// TIA Portal project "PLC1500与G120调速控制" (V14)

(* hardware
DEVICE "S71500/ET200MP station_1"  S7-1500 station
   slot 0: "导轨_0"  Rack  6ES7 590-1***0-0AA0
   slot 1: "Line1_Station1_PLC"  CPU 1516-3 PN/DP  6ES7 516-3AN01-0AB0  V2.1
      slot 3: "CPU 显示_1"  6ES7591-1BA00-0AA0
   slot 2: "DI 32x24VDC HF_1"  DI 32x24VDC HF  6ES7 521-1BL00-0AB0  V2.1
   slot 3: "DQ 32x24VDC/0.5A HF_1"  DQ 32x24VDC/0.5A HF  6ES7 522-1BL01-0AB0  V1.0
   slot 4: "AI 8xU/I/RTD/TC ST_1"  AI 8xU/I/RTD/TC ST  6ES7 531-7KF00-0AB0  V2.1
   slot 5: "AQ 4xU/I ST_1"  AQ 4xU/I ST  6ES7 532-5HD00-0AB0  V2.1
DEVICE "SINAMICS G_1"  Sinamics.Device
   slot 0: "Line1_Station1_G120"  G120 CU250S-2 PN Vector  6SL3246-0BA22-1FA0  4.7.6
   slot 0: "	_0"  Rail
   slot 3: "PM240-2 IP20"  PM240-2 IP20  6SL3210-1PB13-0ULx  -
*)

// ===== PLC "Line1_Station1_PLC"  CPU 1516-3 PN/DP =====

VAR_GLOBAL   // PLC tag table "默认变量表"
   "状态字" AT %IW256 : Word;   // 变频器反馈的状态
   "速度反馈值" AT %IW258 : Word;   // 变频器当前的速度
   "控制字" AT %QW256 : Word;   // PLC控制变频器内容
   "速度设定值" AT %QW258 : Word;   // PLC控制变频器速度
END_VAR

DATA_BLOCK "通讯控制数据"   // DB1
{ S7_Optimized_Access := 'TRUE' }
VERSION : 0.1
   VAR
      启动 : Bool;   // 用于控制驱动启动
      停止 : Bool;   // 用于控制驱动停止
      反转 : Bool;
      复位 : Bool;
      速度反馈值 : Real;   // 用于存放速度反馈值
      速度设定值 : Real;   // 用于存放速度设定值
      临时变量1 : Real;   // 用于过程数据处理临时存放
      临时变量2 : Real;   // 用于过程数据处理临时存放
      临时变量3 : Real;   // 用于过程数据处理临时存放
      临时变量4 : Real;   // 用于过程数据处理临时存放
   END_VAR
BEGIN
END_DATA_BLOCK

ORGANIZATION_BLOCK "Main"   // OB1, LAD, ProgramCycle
TITLE = "Main Program Sweep (Cycle)"
{ S7_Optimized_Access := 'TRUE' }
VERSION : 0.1
   VAR_INPUT
      Initial_Call : Bool;   // Initial call of this OB
      Remanence : Bool;   // =True, if remanent data are available
   END_VAR
BEGIN

REGION Network 1: 启动程序
   // 启动时,把16#047F写到通讯报文控制字
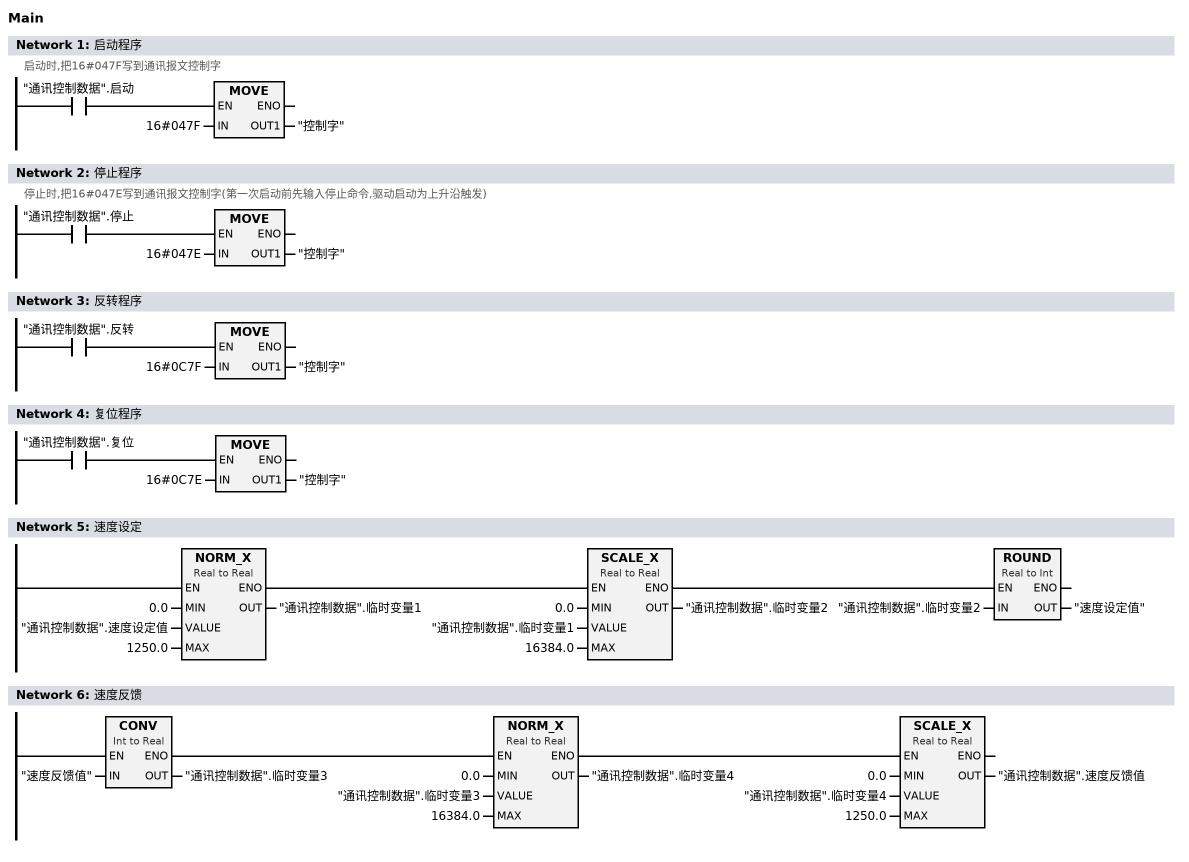
   RUNG wire#powerrail
      Contact( "通讯控制数据".启动 )
      Move(in := 16#047F, out1 => "控制字")
   END_RUNG
   // the same network as SCL:
   IF "通讯控制数据".启动 THEN "控制字" := 16#047F; END_IF;
END_REGION

REGION Network 2: 停止程序
   // 停止时,把16#047E写到通讯报文控制字(第一次启动前先输入停止命令,驱动启动为上升沿触发)
   RUNG wire#powerrail
      Contact( "通讯控制数据".停止 )
      Move(in := 16#047E, out1 => "控制字")
   END_RUNG
   // the same network as SCL:
   IF "通讯控制数据".停止 THEN "控制字" := 16#047E; END_IF;
END_REGION

REGION Network 3: 反转程序
   RUNG wire#powerrail
      Contact( "通讯控制数据".反转 )
      Move(in := 16#0C7F, out1 => "控制字")
   END_RUNG
   // the same network as SCL:
   IF "通讯控制数据".反转 THEN "控制字" := 16#0C7F; END_IF;
END_REGION

REGION Network 4: 复位程序
   RUNG wire#powerrail
      Contact( "通讯控制数据".复位 )
      Move(in := 16#0C7E, out1 => "控制字")
   END_RUNG
   // the same network as SCL:
   IF "通讯控制数据".复位 THEN "控制字" := 16#0C7E; END_IF;
END_REGION

REGION Network 5: 速度设定
   RUNG wire#powerrail
      { S7_Templates := "[SrcType := Real, DestType := Real]" } Normalize(min := 0.0, value := "通讯控制数据".速度设定值, max := 1250.0, out => "通讯控制数据".临时变量1)
      { S7_Templates := "[SrcType := Real, DestType := Real]" } Scale(min := 0.0, value := "通讯控制数据".临时变量1, max := 16384.0, out => "通讯控制数据".临时变量2)
      { S7_Templates := "[SrcType := Real, DestType := Int]" } Round(in := "通讯控制数据".临时变量2, out => "速度设定值")
   END_RUNG
   // the same network as SCL:
   "通讯控制数据".临时变量1 := NORM_X(MIN := 0.0, VALUE := "通讯控制数据".速度设定值, MAX := 1250.0);
   "通讯控制数据".临时变量2 := SCALE_X(MIN := 0.0, VALUE := "通讯控制数据".临时变量1, MAX := 16384.0);
   "速度设定值" := ROUND("通讯控制数据".临时变量2);
END_REGION

REGION Network 6: 速度反馈
   RUNG wire#powerrail
      { S7_Templates := "[SrcType := Int, DestType := Real]" } Convert(in := "速度反馈值", out => "通讯控制数据".临时变量3)
      { S7_Templates := "[SrcType := Real, DestType := Real]" } Normalize(min := 0.0, value := "通讯控制数据".临时变量3, max := 16384.0, out => "通讯控制数据".临时变量4)
      { S7_Templates := "[SrcType := Real, DestType := Real]" } Scale(min := 0.0, value := "通讯控制数据".临时变量4, max := 1250.0, out => "通讯控制数据".速度反馈值)
   END_RUNG
   // the same network as SCL:
   "通讯控制数据".临时变量3 := INT_TO_REAL("速度反馈值");
   "通讯控制数据".临时变量4 := NORM_X(MIN := 0.0, VALUE := "通讯控制数据".临时变量3, MAX := 16384.0);
   "通讯控制数据".速度反馈值 := SCALE_X(MIN := 0.0, VALUE := "通讯控制数据".临时变量4, MAX := 1250.0);
END_REGION
END_ORGANIZATION_BLOCK